// POUs/DIOC/F_GetVersion_FIXSUS_DIOC
FUNCTION F_GetVersion_FIXSUS_DIOC : INT(* Gets the library version info *)
VAR_INPUT
	nVersionElement		:	INT;
(*
	Possible nVersionElement parameter:
	1	:	major number
	2	:	minor number
	3	:	revision number
*)
END_VAR
(* Version history:
Date		|	Version				|	created with					|	Author				|	Remark
dd.mm.yyyy	|						|									|						|
-----------------------------------------------------------------------------------------------------------------------------------------------------------------------------------------------------------------------------------------------------------------------------------
23.12.2016	|	1.0.0				|	TCAT2.11 B2249					|	RK					|	first release
01.03.2017	|	2.0.0				|	TCAT2.11 B2249					|	FixSus				|	Array implementation, FB_Dioc
17.04.2017	|	2.1.0				|	TCAT2.11 B2249					|	RK					|	Library base
01.12.2017	|	3.5.0				|	TCAT2.11 B2259					|	FixSus				|	More generic implementation without arrays
26.01.2018	|	3.6.0				|	TCAT2.11 B2259					|	RK					|	General cleanup for final library and sample
26.01.2018	|	3.7.0				|	TCAT2.11 B2258					|	FixSus (AH)			|	Changed startup timer and visualisation RA
22.03.2018	|	3.8.0				|	TCAT2.11 B2258					|	FixSus (AH)			|	Added comments on visualisation RC
26.03.2018	|	3.9.0				|	TCAT2.11 B2258					|	FixSus (AH/HS)		|	Fixed bugs with DO 45,46 and 47 and added a 1 minute check on the input to know if the island is unplugged.
28.03.2018	|	3.10.0				|	TCAT2.11 B2258					|	FixSus (AH)			|	Added dewpoint calculation to the TP10 and deleted infrared measurements
17.04.2018	|	3.11.0				|	TCAT2.11 B2258					|	FixSus (AH)			| 	Added ForceSend Bools to the RC. If set to true, the analog values will be send immediatly.
19.06.2018	|	3.12.0				| 	TCAT2.11 B2258					|	FixSus (AH)			|	Added input to the TP10 to reset CO2/VOC sensor
19.06.2018	|	3.13.0				| 	TCAT2.11 B2258					|	FixSus (AH)			|	Fixed bug with buffer priority, small change to visualisations and added delay time to the RC startup list.
22.06.2018	|	3.14.0				| 	TCAT2.11 B2258					|	FixSus (AH)			|	VOC/eCO2 values are original sensor values again.
01.07.2018	|	3.15.0				|	TCAT2.11 B2258					|	FixSus (AH)			|	Updated startup timer
02.10.2018	|	3.16.0				|	TCAT2.11 B2258					|	FixSus (AH)			|	Added standard values to RC comments
13.03.2019	|	3.19.0				|	TCAT2.11 B2258					|	FixSus (AH)			|	Added version check to the VOC/eCO2 correction
28.05.2019	|	3.20.0				|	TCAT2.11 B2258					|	FixSus (AH)			|	Fixed startup list bug and sync message is the highest priority message now
30.08.2019	|	3.21.0				|	TCAT2.11 B2258					|	FixSus (AH) 		| 	Deleted reference to the currentvisu variable
12.03.2020	|	3.22.0				|	TCAT2.11 B2259					|	FixSus (AH)			|	RC intervals now use UDINT instead of INTS to avoid overflows with big timing intervals.
20.08.2020	|	3.23.0				|	TCAT2.11 B2277					| 	FixSus (AH)			| 	Completed RC descriptions in english.
27.10.2020	|	3.24.0				|	TCAT2.11 B2277					| 	FixSus (AH)			| 	TP10's with versions between 01/06/2020 and 08/10/2020 will send their temperature offset on a cyclic basis. Also deleted implicit conversions.
26.11.2020	|	3.25.0				|	TCAT2.11 B2277					|	FixSus (AH)			|	Sensitivity is now adjustable through the PLC program
*)

CASE nVersionElement OF
1:	(* major number *)
	F_GetVersion_FIXSUS_DIOC := 3;
2:	(* minor number *)
	F_GetVersion_FIXSUS_DIOC := 25;
3:	(* revision number *)
	F_GetVersion_FIXSUS_DIOC := 0;
ELSE
	F_GetVersion_FIXSUS_DIOC := -1;
END_CASE

END_FUNCTION

// Visualizations/DIOC/RC/RC_PARTS/RC_FP
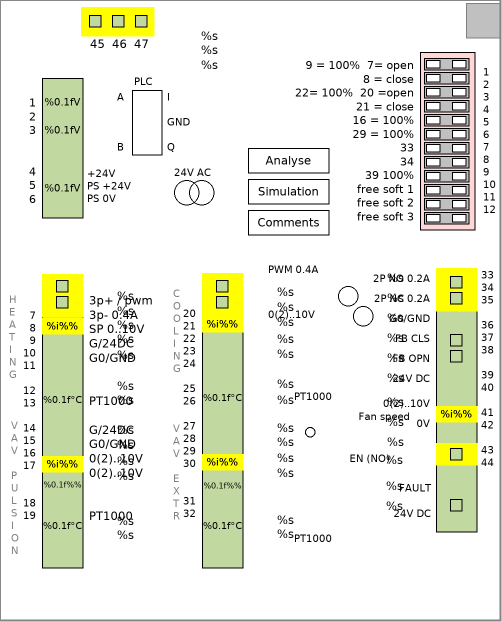
VISUALIZATION RC_FP  // 502x622
VAR_IN_OUT
	m_Input_GROUP : None;
END_VAR
    Rectangle (0,0 500x620)
    Rectangle (81,7 72x28)
    Rectangle (81,7 73x29), invisible if: NOT m_Input_GROUP._bSim, input disabled if: NOT m_Input_GROUP._bSim
    Rectangle (202,274 41x294)
    Rectangle (436,268 41x264)
    Rectangle (202,273 41x43), invisible if: NOT m_Input_GROUP._bSim, input disabled if: NOT m_Input_GROUP._bSim
    Rectangle (436,268 41x43), invisible if: NOT m_Input_GROUP._bSim, input disabled if: NOT m_Input_GROUP._bSim
    Rectangle (436,443 41x22), invisible if: NOT m_Input_GROUP._bSim, input disabled if: NOT m_Input_GROUP._bSim
    Rectangle (42,274 41x294)
    Rectangle (42,274 41x43), invisible if: NOT m_Input_GROUP._bSim, input disabled if: NOT m_Input_GROUP._bSim
    Polyline (133,133)
    Polyline (72,112)
    Rectangle (262,46 155x190), "9 = 100% 7= open 8 = close 22= 100% 20 =open 21 = close 16 = 100% 29 = 100% 33 34 39 100% free soft 1 free soft 2 free soft 3"
    Rectangle (24,268 15x295), "7 8 9 10 11 12 13 14 15 16 17 18 19"
    Rectangle (86,268 90x295), "3p+ / pwm 3p- 0.4A SP 0..10V G/24DC G0/GND PT1000 G/24DC G0/GND 0(2)..10V 0(2)..10V PT1000", invisible if: (m_Input_GROUP._bComments) <> 0
    Rectangle (184,266 15x295), "20 21 22 23 24 25 26 27 28 29 30 31 32"
    Rectangle (6,272 10x130), "H E A T I N G"
    Rectangle (8,416 10x144), "V A V P U L S I O N"
    Rectangle (170,411 10x135), "V A V E X T R"
    Rectangle (170,266 10x130), "C O O L I N G"
    Rectangle (42,392 41x16), "%0.1f°C", text variable: m_Input_GROUP.qfTempHeatingWater
    Rectangle (42,518 41x16), "%0.1f°C", text variable: m_Input_GROUP.qfTempAirPulsion
    Rectangle (42,318 41x16), "%i%%", text variable: m_Input_GROUP._iSpHeatingSim, invisible if: NOT m_Input_GROUP._bSim, input disabled if: NOT m_Input_GROUP._bSim
        OnMouseDown: write the text variable via VisuDialogs.Numpad, min 0, max 100
    Rectangle (42,456 41x16), "%i%%", text variable: m_Input_GROUP._iSpPulsionSim, invisible if: NOT m_Input_GROUP._bSim, input disabled if: NOT m_Input_GROUP._bSim
        OnMouseDown: write the text variable via VisuDialogs.Numpad, min 0, max 100
    Rectangle (42,477 41x16), "%0.1f%%", text variable: m_Input_GROUP.qfPulsionFB
    Rectangle (56,280 12x12), colour toggle: (m_Input_GROUP.bHeating_3P_plus) <> 0, invisible if: (m_Input_GROUP._bSim) <> 0, input disabled if: (m_Input_GROUP._bSim) <> 0
    Rectangle (56,296 12x12), colour toggle: (m_Input_GROUP.bHeating_3P_min) <> 0, invisible if: (m_Input_GROUP._bSim) <> 0, input disabled if: (m_Input_GROUP._bSim) <> 0
    Rectangle (202,390 41x16), "%0.1f°C", text variable: m_Input_GROUP.qfTempIceWater
    Rectangle (202,518 41x16), "%0.1f°C", text variable: m_Input_GROUP.qfTempAirExtraction
    Rectangle (202,316 41x16), "%i%%", text variable: m_Input_GROUP._iSpCoolingSim, invisible if: NOT m_Input_GROUP._bSim, input disabled if: NOT m_Input_GROUP._bSim
        OnMouseDown: write the text variable via VisuDialogs.Numpad, min 0, max 100
    Rectangle (202,454 41x16), "%i%%", text variable: m_Input_GROUP._iSpExtractionSim, invisible if: NOT m_Input_GROUP._bSim, input disabled if: NOT m_Input_GROUP._bSim
        OnMouseDown: write the text variable via VisuDialogs.Numpad, min 0, max 100
    Rectangle (202,478 41x16), "%0.1f%%", text variable: m_Input_GROUP.qfExtractionFB
    Rectangle (216,296 12x12), colour toggle: (m_Input_GROUP._bCooling_3P_minSim) <> 0, invisible if: NOT m_Input_GROUP._bSim, input disabled if: NOT m_Input_GROUP._bSim
        toggle m_Input_GROUP._bCooling_3P_minSim
    Rectangle (216,280 12x12), colour toggle: (m_Input_GROUP._bCooling_3P_plusSim) <> 0, invisible if: NOT m_Input_GROUP._bSim, input disabled if: NOT m_Input_GROUP._bSim
        toggle m_Input_GROUP._bCooling_3P_plusSim
    Rectangle (478,268 15x295), "33 34 35 36 37 38 39 40 41 42 43 44"
    Rectangle (436,406 41x16), "%i%%", text variable: m_Input_GROUP._iSpFanSim, invisible if: NOT m_Input_GROUP._bSim, input disabled if: NOT m_Input_GROUP._bSim
        OnMouseDown: write the text variable via VisuDialogs.Numpad, min 0, max 100
    Rectangle (450,276 12x12), colour toggle: (m_Input_GROUP._bFireDamper_OPNSim) <> 0, invisible if: NOT m_Input_GROUP._bSim, input disabled if: NOT m_Input_GROUP._bSim
        toggle m_Input_GROUP._bFireDamper_OPNSim
    Rectangle (450,292 12x12), colour toggle: (m_Input_GROUP._bFireDamper_CLSSim) <> 0, invisible if: NOT m_Input_GROUP._bSim, input disabled if: NOT m_Input_GROUP._bSim
        toggle m_Input_GROUP._bFireDamper_CLSSim
    Rectangle (450,350 12x12), colour toggle: (m_Input_GROUP.qbFireDamperFB_OPN) <> 0
    Rectangle (450,334 12x12), colour toggle: (m_Input_GROUP.qbFireDamperFB_CLS) <> 0
    Rectangle (450,448 12x12), colour toggle: (m_Input_GROUP._bEnableFanSim) <> 0, invisible if: NOT m_Input_GROUP._bSim, input disabled if: NOT m_Input_GROUP._bSim
        toggle m_Input_GROUP._bEnableFanSim
    Rectangle (24,83 15x150), "1 2 3 4 5 6"
    Rectangle (42,78 41x140)
    Rectangle (42,180 41x16), "%0.1fV", text variable: m_Input_GROUP.qfACVoltageLevel
    Rectangle (42,94 41x16), "%0.1fV", text variable: m_Input_GROUP.qrVoltageLevelA
    Rectangle (42,122 41x16), "%0.1fV", text variable: m_Input_GROUP.qrVoltageLevelB
    Rectangle (420,52 55x178)
    Rectangle (480,46 15x190), "1 2 3 4 5 6 7 8 9 10 11 12"
    Frame (424,58 47x14)
        shows UDO_DIPSWITCH(m_Input_GROUP := m_Input_GROUP, m_Input_ON_SIGNAAL := qarr_bDipSwitches[1])
    Frame (424,72 47x14)
        shows UDO_DIPSWITCH(m_Input_GROUP := m_Input_GROUP, m_Input_ON_SIGNAAL := qarr_bDipSwitches[2])
    Frame (424,86 47x14)
        shows UDO_DIPSWITCH(m_Input_GROUP := m_Input_GROUP, m_Input_ON_SIGNAAL := qarr_bDipSwitches[3])
    Frame (424,100 47x14)
        shows UDO_DIPSWITCH(m_Input_GROUP := m_Input_GROUP, m_Input_ON_SIGNAAL := qarr_bDipSwitches[4])
    Frame (424,114 47x14)
        shows UDO_DIPSWITCH(m_Input_GROUP := m_Input_GROUP, m_Input_ON_SIGNAAL := qarr_bDipSwitches[5])
    Frame (424,128 47x14)
        shows UDO_DIPSWITCH(m_Input_GROUP := m_Input_GROUP, m_Input_ON_SIGNAAL := qarr_bDipSwitches[6])
    Frame (424,142 47x14)
        shows UDO_DIPSWITCH(m_Input_GROUP := m_Input_GROUP, m_Input_ON_SIGNAAL := qarr_bDipSwitches[7])
    Frame (424,156 47x14)
        shows UDO_DIPSWITCH(m_Input_GROUP := m_Input_GROUP, m_Input_ON_SIGNAAL := qarr_bDipSwitches[8])
    Frame (424,170 47x14)
        shows UDO_DIPSWITCH(m_Input_GROUP := m_Input_GROUP, m_Input_ON_SIGNAAL := qarr_bDipSwitches[9])
    Frame (424,184 47x14)
        shows UDO_DIPSWITCH(m_Input_GROUP := m_Input_GROUP, m_Input_ON_SIGNAAL := qarr_bDipSwitches[10])
    Frame (424,198 47x14)
        shows UDO_DIPSWITCH(m_Input_GROUP := m_Input_GROUP, m_Input_ON_SIGNAAL := qarr_bDipSwitches[11])
    Frame (424,212 47x14)
        shows UDO_DIPSWITCH(m_Input_GROUP := m_Input_GROUP, m_Input_ON_SIGNAAL := qarr_bDipSwitches[12])
    Polyline (224,185)
    Polyline (224,200)
    Rectangle (132,90 30x65)
    Polyline (177,200)
    Polyline (164,210)
    Polyline (168,210)
    Ellipse (174,180 25x25)
    Ellipse (189,180 25x25)
    Rectangle (96,82 31x80), "A B"
    Rectangle (164,82 30x80), "I GND Q"
    Rectangle (131,74 40x15), "PLC"
    Rectangle (84,146 65x80), "+24V PS +24V PS 0V"
    Rectangle (144,165 70x15), "24V AC"
    Polyline (133,187)
    Polyline (111,171)
    Rectangle (248,179 81x25), "Simulation"
        toggle m_Input_GROUP._bSim
    Rectangle (56,280 12x12), colour toggle: (m_Input_GROUP._bHeating_3P_plusSim) <> 0, invisible if: NOT m_Input_GROUP._bSim, input disabled if: NOT m_Input_GROUP._bSim
        toggle m_Input_GROUP._bHeating_3P_plusSim
    Rectangle (56,296 12x12), colour toggle: (m_Input_GROUP._bHeating_3P_minSim) <> 0, invisible if: NOT m_Input_GROUP._bSim, input disabled if: NOT m_Input_GROUP._bSim
        toggle m_Input_GROUP._bHeating_3P_minSim
    Rectangle (42,318 41x16), "%i%%", text variable: m_Input_GROUP.iSpHeating, invisible if: (m_Input_GROUP._bSim) <> 0, input disabled if: (m_Input_GROUP._bSim) <> 0
    Rectangle (42,456 41x16), "%i%%", text variable: m_Input_GROUP.iSpPulsion, invisible if: (m_Input_GROUP._bSim) <> 0, input disabled if: (m_Input_GROUP._bSim) <> 0
    Rectangle (202,316 41x16), "%i%%", text variable: m_Input_GROUP.iSpCooling, invisible if: (m_Input_GROUP._bSim) <> 0, input disabled if: (m_Input_GROUP._bSim) <> 0
    Rectangle (202,454 41x16), "%i%%", text variable: m_Input_GROUP.iSpExtraction, invisible if: (m_Input_GROUP._bSim) <> 0, input disabled if: (m_Input_GROUP._bSim) <> 0
    Rectangle (216,296 12x12), colour toggle: (m_Input_GROUP.bCooling_3P_min) <> 0, invisible if: (m_Input_GROUP._bSim) <> 0, input disabled if: (m_Input_GROUP._bSim) <> 0
    Rectangle (216,280 12x12), colour toggle: (m_Input_GROUP.bCooling_3P_plus) <> 0, invisible if: (m_Input_GROUP._bSim) <> 0, input disabled if: (m_Input_GROUP._bSim) <> 0
    Rectangle (436,406 41x16), "%i%%", text variable: m_Input_GROUP.iSpFan, invisible if: (m_Input_GROUP._bSim) <> 0, input disabled if: (m_Input_GROUP._bSim) <> 0
    Rectangle (450,276 12x12), colour toggle: (m_Input_GROUP.bFireDamper_OPN) <> 0, invisible if: (m_Input_GROUP._bSim) <> 0, input disabled if: (m_Input_GROUP._bSim) <> 0
    Rectangle (450,292 12x12), colour toggle: (m_Input_GROUP.bFireDamper_CLS) <> 0, invisible if: (m_Input_GROUP._bSim) <> 0, input disabled if: (m_Input_GROUP._bSim) <> 0
    Rectangle (450,448 12x12), colour toggle: (m_Input_GROUP.bEnableFan) <> 0, invisible if: (m_Input_GROUP._bSim) <> 0, input disabled if: (m_Input_GROUP._bSim) <> 0
    Rectangle (450,499 12x12), colour toggle: (m_Input_GROUP.qbFanFault) <> 0
    Group (466,3 32x33)
        toggle m_Input_GROUP._bSelected
        RoundedRectangle (0,0 34x35)
        Polyline (28,28)
        Polyline (7,28)
    Rectangle (87,38 74x12), "45 46 47", invisible if: (m_Input_GROUP._bComments) <> 0
    Rectangle (89,15 12x12), colour toggle: (m_Input_GROUP.bRelais_45) <> 0, invisible if: (m_Input_GROUP._bSim) <> 0, input disabled if: (m_Input_GROUP._bSim) <> 0
    Rectangle (112,15 12x12), colour toggle: (m_Input_GROUP.bRelais_46) <> 0, invisible if: (m_Input_GROUP._bSim) <> 0, input disabled if: (m_Input_GROUP._bSim) <> 0
    Rectangle (135,15 12x12), colour toggle: (m_Input_GROUP.bRelais_47) <> 0, invisible if: (m_Input_GROUP._bSim) <> 0, input disabled if: (m_Input_GROUP._bSim) <> 0
    Rectangle (89,15 12x12), colour toggle: (m_Input_GROUP._bRelais_45Sim) <> 0, invisible if: NOT m_Input_GROUP._bSim, input disabled if: NOT m_Input_GROUP._bSim
        toggle m_Input_GROUP._bRelais_45Sim
    Rectangle (112,15 12x12), colour toggle: (m_Input_GROUP._bRelais_46Sim) <> 0, invisible if: NOT m_Input_GROUP._bSim, input disabled if: NOT m_Input_GROUP._bSim
        toggle m_Input_GROUP._bRelais_46Sim
    Rectangle (135,15 12x12), colour toggle: (m_Input_GROUP._bRelais_47Sim) <> 0, invisible if: NOT m_Input_GROUP._bSim, input disabled if: NOT m_Input_GROUP._bSim
        toggle m_Input_GROUP._bRelais_47Sim
    Rectangle (248,148 81x25), "Analyse", invisible if: NOT Global_DIOC_Variables_Debug.DIOC_Debug, input disabled if: NOT Global_DIOC_Variables_Debug.DIOC_Debug
        toggle m_Input_GROUP._bAnalyse
    Rectangle (248,210 81x25), "Comments"
        toggle m_Input_GROUP._bComments
    Group (245,262 192x291), invisible if: (m_Input_GROUP._bComments) <> 0
        Polyline (0,30)
        Polyline (0,105)
        Polyline (70,40)
        Polyline (70,30)
        Polyline (70,25)
        Polyline (70,35)
        Polyline (40,65)
        Polyline (40,70)
        Polyline (30,105)
        Group (26,6 18x33)
            Polygon (20,20)
            Polyline (20,20)
        Group (41,51 18x33)
            Polygon (20,20)
            Polyline (20,20)
        Polyline (40,120)
        Polyline (40,145)
        Polyline (40,263)
        Polyline (40,288)
        Polyline (50,214)
        Polyline (50,195)
        Polyline (50,205)
        Polyline (50,215)
        Polyline (80,180)
        Ellipse (60,165 10x10)
        Ellipse (93,24 20x20)
        Rectangle (20,0 60x15), "PWM 0.4A"
        Rectangle (20,45 60x15), "0(2)..10V"
        Rectangle (46,127 60x15), "PT1000"
        Rectangle (46,269 60x15), "PT1000"
        Ellipse (108,44 20x20)
        Polyline (193,24)
        Polyline (193,44)
        Polyline (193,64)
        Polyline (118,69)
        Polyline (193,124)
        Polyline (118,79)
        Polyline (118,99)
        Polyline (133,149)
        Polyline (133,169)
        Polyline (163,189)
        Polyline (118,204)
        Polyline (168,194)
        Polyline (178,189)
        Polyline (124,224)
        Polyline (194,259)
        Rectangle (118,9 70x15), "2P NO 0.2A"
        Rectangle (118,29 70x15), "2P NC 0.2A"
        Rectangle (118,49 70x15), "G0/GND"
        Rectangle (118,69 70x15), "FB CLS"
        Rectangle (118,89 70x15), "FB OPN"
        Rectangle (118,109 70x15), "24V DC"
        Rectangle (118,134 70x15), "0(2)..10V"
        Rectangle (98,147 70x15), "Fan speed"
        Rectangle (118,154 70x15), "0V"
        Rectangle (78,189 70x15), "EN (NO)"
        Rectangle (119,219 70x14), "FAULT"
        Rectangle (119,244 70x15), "24V DC"
        Polyline (50,215)
        Polyline (103,104)
        Polyline (17,220)
        Polyline (5,201)
    Rectangle (84,289 83x14), "%s", text variable: m_Input_GROUP.arr_sConnectionComments[1], invisible if: NOT m_Input_GROUP._bComments, input disabled if: NOT m_Input_GROUP._bComments
        OnMouseDown: write the text variable via Edit
    Rectangle (84,304 83x14), "%s", text variable: m_Input_GROUP.arr_sConnectionComments[2], invisible if: NOT m_Input_GROUP._bComments, input disabled if: NOT m_Input_GROUP._bComments
        OnMouseDown: write the text variable via Edit
    Rectangle (84,318 83x14), "%s", text variable: m_Input_GROUP.arr_sConnectionComments[3], invisible if: NOT m_Input_GROUP._bComments, input disabled if: NOT m_Input_GROUP._bComments
        OnMouseDown: write the text variable via Edit
    Rectangle (84,332 83x14), "%s", text variable: m_Input_GROUP.arr_sConnectionComments[4], invisible if: NOT m_Input_GROUP._bComments, input disabled if: NOT m_Input_GROUP._bComments
        OnMouseDown: write the text variable via Edit
    Rectangle (84,348 83x14), "%s", text variable: m_Input_GROUP.arr_sConnectionComments[5], invisible if: NOT m_Input_GROUP._bComments, input disabled if: NOT m_Input_GROUP._bComments
        OnMouseDown: write the text variable via Edit
    Rectangle (84,379 83x14), "%s", text variable: m_Input_GROUP.arr_sConnectionComments[6], invisible if: NOT m_Input_GROUP._bComments, input disabled if: NOT m_Input_GROUP._bComments
        OnMouseDown: write the text variable via Edit
    Rectangle (84,393 83x14), "%s", text variable: m_Input_GROUP.arr_sConnectionComments[7], invisible if: NOT m_Input_GROUP._bComments, input disabled if: NOT m_Input_GROUP._bComments
        OnMouseDown: write the text variable via Edit
    Rectangle (84,423 83x14), "%s", text variable: m_Input_GROUP.arr_sConnectionComments[8], invisible if: NOT m_Input_GROUP._bComments, input disabled if: NOT m_Input_GROUP._bComments
        OnMouseDown: write the text variable via Edit
    Rectangle (84,438 83x14), "%s", text variable: m_Input_GROUP.arr_sConnectionComments[9], invisible if: NOT m_Input_GROUP._bComments, input disabled if: NOT m_Input_GROUP._bComments
        OnMouseDown: write the text variable via Edit
    Rectangle (84,454 83x14), "%s", text variable: m_Input_GROUP.arr_sConnectionComments[10], invisible if: NOT m_Input_GROUP._bComments, input disabled if: NOT m_Input_GROUP._bComments
        OnMouseDown: write the text variable via Edit
    Rectangle (84,469 83x14), "%s", text variable: m_Input_GROUP.arr_sConnectionComments[11], invisible if: NOT m_Input_GROUP._bComments, input disabled if: NOT m_Input_GROUP._bComments
        OnMouseDown: write the text variable via Edit
    Rectangle (84,514 83x14), "%s", text variable: m_Input_GROUP.arr_sConnectionComments[12], invisible if: NOT m_Input_GROUP._bComments, input disabled if: NOT m_Input_GROUP._bComments
        OnMouseDown: write the text variable via Edit
    Rectangle (84,528 83x14), "%s", text variable: m_Input_GROUP.arr_sConnectionComments[13], invisible if: NOT m_Input_GROUP._bComments, input disabled if: NOT m_Input_GROUP._bComments
        OnMouseDown: write the text variable via Edit
    Rectangle (244,285 83x14), "%s", text variable: m_Input_GROUP.arr_sConnectionComments[14], invisible if: NOT m_Input_GROUP._bComments, input disabled if: NOT m_Input_GROUP._bComments
        OnMouseDown: write the text variable via Edit
    Rectangle (244,300 83x14), "%s", text variable: m_Input_GROUP.arr_sConnectionComments[15], invisible if: NOT m_Input_GROUP._bComments, input disabled if: NOT m_Input_GROUP._bComments
        OnMouseDown: write the text variable via Edit
    Rectangle (244,315 83x14), "%s", text variable: m_Input_GROUP.arr_sConnectionComments[16], invisible if: NOT m_Input_GROUP._bComments, input disabled if: NOT m_Input_GROUP._bComments
        OnMouseDown: write the text variable via Edit
    Rectangle (244,332 83x14), "%s", text variable: m_Input_GROUP.arr_sConnectionComments[17], invisible if: NOT m_Input_GROUP._bComments, input disabled if: NOT m_Input_GROUP._bComments
        OnMouseDown: write the text variable via Edit
    Rectangle (244,347 83x14), "%s", text variable: m_Input_GROUP.arr_sConnectionComments[18], invisible if: NOT m_Input_GROUP._bComments, input disabled if: NOT m_Input_GROUP._bComments
        OnMouseDown: write the text variable via Edit
    Rectangle (244,377 83x14), "%s", text variable: m_Input_GROUP.arr_sConnectionComments[19], invisible if: NOT m_Input_GROUP._bComments, input disabled if: NOT m_Input_GROUP._bComments
        OnMouseDown: write the text variable via Edit
    Rectangle (244,393 83x14), "%s", text variable: m_Input_GROUP.arr_sConnectionComments[20], invisible if: NOT m_Input_GROUP._bComments, input disabled if: NOT m_Input_GROUP._bComments
        OnMouseDown: write the text variable via Edit
    Rectangle (244,421 83x14), "%s", text variable: m_Input_GROUP.arr_sConnectionComments[21], invisible if: NOT m_Input_GROUP._bComments, input disabled if: NOT m_Input_GROUP._bComments
        OnMouseDown: write the text variable via Edit
    Rectangle (244,435 83x14), "%s", text variable: m_Input_GROUP.arr_sConnectionComments[22], invisible if: NOT m_Input_GROUP._bComments, input disabled if: NOT m_Input_GROUP._bComments
        OnMouseDown: write the text variable via Edit
    Rectangle (244,451 83x14), "%s", text variable: m_Input_GROUP.arr_sConnectionComments[23], invisible if: NOT m_Input_GROUP._bComments, input disabled if: NOT m_Input_GROUP._bComments
        OnMouseDown: write the text variable via Edit
    Rectangle (244,466 83x14), "%s", text variable: m_Input_GROUP.arr_sConnectionComments[24], invisible if: NOT m_Input_GROUP._bComments, input disabled if: NOT m_Input_GROUP._bComments
        OnMouseDown: write the text variable via Edit
    Rectangle (244,513 83x14), "%s", text variable: m_Input_GROUP.arr_sConnectionComments[25], invisible if: NOT m_Input_GROUP._bComments, input disabled if: NOT m_Input_GROUP._bComments
        OnMouseDown: write the text variable via Edit
    Rectangle (244,527 83x14), "%s", text variable: m_Input_GROUP.arr_sConnectionComments[26], invisible if: NOT m_Input_GROUP._bComments, input disabled if: NOT m_Input_GROUP._bComments
        OnMouseDown: write the text variable via Edit
    Rectangle (354,271 83x14), "%s", text variable: m_Input_GROUP.arr_sConnectionComments[27], invisible if: NOT m_Input_GROUP._bComments, input disabled if: NOT m_Input_GROUP._bComments
        OnMouseDown: write the text variable via Edit
    Rectangle (354,291 83x14), "%s", text variable: m_Input_GROUP.arr_sConnectionComments[28], invisible if: NOT m_Input_GROUP._bComments, input disabled if: NOT m_Input_GROUP._bComments
        OnMouseDown: write the text variable via Edit
    Rectangle (354,311 83x14), "%s", text variable: m_Input_GROUP.arr_sConnectionComments[29], invisible if: NOT m_Input_GROUP._bComments, input disabled if: NOT m_Input_GROUP._bComments
        OnMouseDown: write the text variable via Edit
    Rectangle (354,331 83x14), "%s", text variable: m_Input_GROUP.arr_sConnectionComments[30], invisible if: NOT m_Input_GROUP._bComments, input disabled if: NOT m_Input_GROUP._bComments
        OnMouseDown: write the text variable via Edit
    Rectangle (354,351 83x14), "%s", text variable: m_Input_GROUP.arr_sConnectionComments[31], invisible if: NOT m_Input_GROUP._bComments, input disabled if: NOT m_Input_GROUP._bComments
        OnMouseDown: write the text variable via Edit
    Rectangle (354,371 83x14), "%s", text variable: m_Input_GROUP.arr_sConnectionComments[32], invisible if: NOT m_Input_GROUP._bComments, input disabled if: NOT m_Input_GROUP._bComments
        OnMouseDown: write the text variable via Edit
    Rectangle (354,395 83x14), "%s", text variable: m_Input_GROUP.arr_sConnectionComments[33], invisible if: NOT m_Input_GROUP._bComments, input disabled if: NOT m_Input_GROUP._bComments
        OnMouseDown: write the text variable via Edit
    Rectangle (354,415 83x14), "%s", text variable: m_Input_GROUP.arr_sConnectionComments[34], invisible if: NOT m_Input_GROUP._bComments, input disabled if: NOT m_Input_GROUP._bComments
        OnMouseDown: write the text variable via Edit
    Rectangle (354,435 83x14), "%s", text variable: m_Input_GROUP.arr_sConnectionComments[35], invisible if: NOT m_Input_GROUP._bComments, input disabled if: NOT m_Input_GROUP._bComments
        OnMouseDown: write the text variable via Edit
    Rectangle (353,453 83x14), "%s", text variable: m_Input_GROUP.arr_sConnectionComments[36], invisible if: NOT m_Input_GROUP._bComments, input disabled if: NOT m_Input_GROUP._bComments
        OnMouseDown: write the text variable via Edit
    Rectangle (353,479 83x14), "%s", text variable: m_Input_GROUP.arr_sConnectionComments[37], invisible if: NOT m_Input_GROUP._bComments, input disabled if: NOT m_Input_GROUP._bComments
        OnMouseDown: write the text variable via Edit
    Rectangle (353,499 83x14), "%s", text variable: m_Input_GROUP.arr_sConnectionComments[38], invisible if: NOT m_Input_GROUP._bComments, input disabled if: NOT m_Input_GROUP._bComments
        OnMouseDown: write the text variable via Edit
    Rectangle (168,29 83x14), "%s", text variable: m_Input_GROUP.arr_sConnectionComments[39], invisible if: NOT m_Input_GROUP._bComments, input disabled if: NOT m_Input_GROUP._bComments
        OnMouseDown: write the text variable via Edit
    Rectangle (168,43 83x14), "%s", text variable: m_Input_GROUP.arr_sConnectionComments[40], invisible if: NOT m_Input_GROUP._bComments, input disabled if: NOT m_Input_GROUP._bComments
        OnMouseDown: write the text variable via Edit
    Rectangle (168,58 83x14), "%s", text variable: m_Input_GROUP.arr_sConnectionComments[41], invisible if: NOT m_Input_GROUP._bComments, input disabled if: NOT m_Input_GROUP._bComments
        OnMouseDown: write the text variable via Edit
    Polyline (190,45), invisible if: NOT m_Input_GROUP._bComments
    Polyline (190,56), invisible if: NOT m_Input_GROUP._bComments
    Polyline (190,68), invisible if: NOT m_Input_GROUP._bComments
END_VISUALIZATION

// Visualizations/DIOC/RC/RC_PARTS/RC_ROOM_ICON
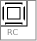
VISUALIZATION RC_ROOM_ICON  // 37x41
    Rectangle (0,0 27x26)
    Rectangle (7,7 13x12)
    Rectangle (5,3 17x0)
    Rectangle (5,23 17x0)
    Rectangle (24,6 0x14)
    Rectangle (3,6 0x14)
    Rectangle (-10,26 45x13), "RC"
    Rectangle (-2,0 30x25)
END_VISUALIZATION

// Visualizations/DIOC/RC/RC_PARTS/UDO_DIPSWITCH
VISUALIZATION UDO_DIPSWITCH  // 47x14
VAR_INPUT
	m_Input_GROUP : None;
END_VAR
VAR_INPUT
	m_Input_ON_SIGNAAL : None;
END_VAR
    Rectangle (0,0 45x12)
    Rectangle (28,2 14x8), invisible if: NOT m_Input_GROUP.m_Input_ON_SIGNAAL
    Rectangle (2,2 14x8), invisible if: ((m_Input_GROUP.m_Input_ON_SIGNAAL)) <> 0
END_VISUALIZATION

// Visualizations/DIOC/RC/RC
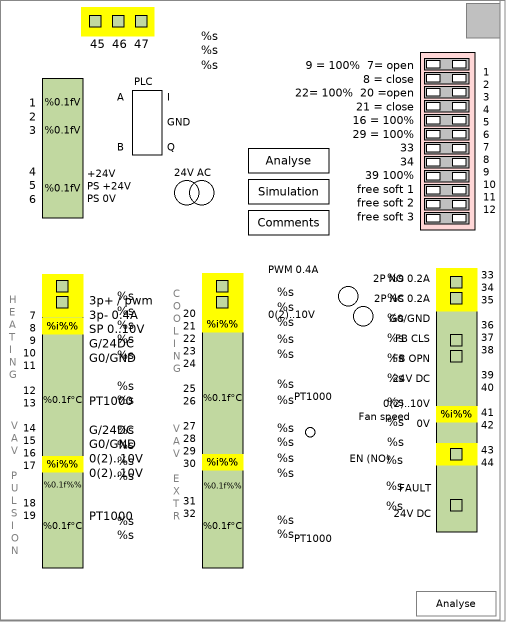
VISUALIZATION RC  // 506x622
VAR_IN_OUT
	m_Input_FB_RC : None;
END_VAR
VAR_IN_OUT
	m_Input_GROUP : None;
END_VAR
VAR_IN_OUT
	m_Input_AnalyseScherm : None;
END_VAR
    Frame (0,0 504x620)
        shows RC_FP(m_Input_GROUP := m_Input_FB_RC)
    Rectangle (416,591 80x25), "Analyse", invisible if: NOT Global_DIOC_Variables_Debug.DIOC_Debug, input disabled if: NOT Global_DIOC_Variables_Debug.DIOC_Debug
        toggle m_Input_GROUP._bAnalyse
END_VISUALIZATION

// Visualizations/DIOC/RC/RC_MINI
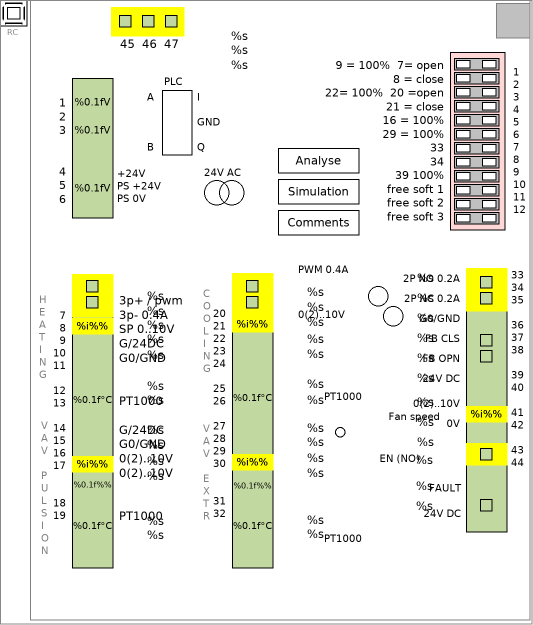
VISUALIZATION RC_MINI  // 533x625
VAR_IN_OUT
	m_Input_FB_RC : None;
END_VAR
VAR_IN_OUT
	m_Input_X_OFFSET : None;
END_VAR
VAR_IN_OUT
	m_Input_Y_OFFSET : None;
END_VAR
    Frame (0,0 27x33)
        shows RC_ROOM_ICON()
        toggle m_Input_FB_RC._bSelected
    Frame (30,0 501x623), invisible if: NOT (m_Input_FB_RC._bSelected), input disabled if: NOT (m_Input_FB_RC._bSelected)
        shows RC_FP(m_Input_GROUP := m_Input_FB_RC)
        p3560616238: m_Input_X_OFFSET
        p2738717112: m_Input_Y_OFFSET
END_VISUALIZATION

// Visualizations/DIOC/TP10/TP10_PARTS/TP10_FP
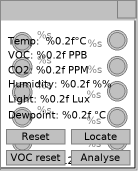
VISUALIZATION TP10_FP  // 138x171
VAR_IN_OUT
	m_Input_GROUP : None;
END_VAR
    Rectangle (0,18 135x150)
    Rectangle (0,-2 135x170)
    Rectangle (0,-2 135x22)
    Polygon (85,13), invisible if: (m_Input_GROUP.bRoomAnalyser) <> 0, input disabled if: (m_Input_GROUP.bRoomAnalyser) <> 0
    Polygon (99,13), invisible if: (m_Input_GROUP.bRoomAnalyser) <> 0, input disabled if: (m_Input_GROUP.bRoomAnalyser) <> 0
    Rectangle (92,-1 22x19), invisible if: (m_Input_GROUP.bRoomAnalyser) <> 0, input disabled if: (m_Input_GROUP.bRoomAnalyser) <> 0
        toggle m_Input_GROUP._bNextVisu
    Group (117,-1 17x17)
        toggle m_Input_GROUP._bSelected
        RoundedRectangle (0,0 19x19)
        Polyline (15,15)
        Polyline (3,15)
    Rectangle (68,0 22x19), invisible if: (m_Input_GROUP.bRoomAnalyser) <> 0, input disabled if: (m_Input_GROUP.bRoomAnalyser) <> 0
        toggle m_Input_GROUP._bPrevVisu
    Group (3,23 130x144), invisible if: m_Input_GROUP._iVis <> 0, input disabled if: m_Input_GROUP._iVis <> 0
        Rectangle (0,129 132x17), "%0.2f°C", text variable: m_Input_GROUP.qfRoomTemperature
        Group (8,101 78x26)
            Ellipse (1,8 20x20), colour variable: m_Input_GROUP._dwVisColor
            Ellipse (3,10 16x16), colour toggle: (m_Input_GROUP.arr_bLeds[5]) <> 0
            Rectangle (23,0 57x22), "%s", text variable: m_Input_GROUP.arr_sButtonComments[5]
            Rectangle (0,7 51x21), invisible if: (m_Input_GROUP.arr_bMasks[5]) <> 0, input disabled if: (m_Input_GROUP.arr_bMasks[5]) <> 0
                tap m_Input_GROUP._arr_bVisuButtons[5]
        Group (8,76 78x26)
            Ellipse (1,8 20x20), colour variable: m_Input_GROUP._dwVisColor
            Ellipse (3,10 16x16), colour toggle: (m_Input_GROUP.arr_bLeds[4]) <> 0
            Rectangle (23,0 57x22), "%s", text variable: m_Input_GROUP.arr_sButtonComments[4]
            Rectangle (0,7 51x21), invisible if: (m_Input_GROUP.arr_bMasks[4]) <> 0, input disabled if: (m_Input_GROUP.arr_bMasks[4]) <> 0
                tap m_Input_GROUP._arr_bVisuButtons[4]
        Group (9,51 77x26)
            Ellipse (0,8 20x20), colour variable: m_Input_GROUP._dwVisColor
            Ellipse (2,10 16x16), colour toggle: (m_Input_GROUP.arr_bLeds[3]) <> 0
            Rectangle (22,0 57x22), "%s", text variable: m_Input_GROUP.arr_sButtonComments[3]
            Rectangle (0,7 51x21), invisible if: (m_Input_GROUP.arr_bMasks[3]) <> 0, input disabled if: (m_Input_GROUP.arr_bMasks[3]) <> 0
                tap m_Input_GROUP._arr_bVisuButtons[3]
        Group (9,26 77x26)
            Ellipse (0,8 20x20), colour variable: m_Input_GROUP._dwVisColor
            Ellipse (2,10 16x16), colour toggle: (m_Input_GROUP.arr_bLeds[2]) <> 0
            Rectangle (22,0 57x22), "%s", text variable: m_Input_GROUP.arr_sButtonComments[2]
            Rectangle (0,7 51x21), invisible if: (m_Input_GROUP.arr_bMasks[2]) <> 0, input disabled if: (m_Input_GROUP.arr_bMasks[2]) <> 0
                tap m_Input_GROUP._arr_bVisuButtons[2]
        Group (46,7 78x23)
            Ellipse (58,0 20x20), colour variable: m_Input_GROUP._dwVisColor
            Ellipse (60,2 16x16), colour toggle: (m_Input_GROUP.arr_bLeds[6]) <> 0
            Rectangle (0,2 56x23), "%s", text variable: m_Input_GROUP.arr_sButtonComments[6]
            Rectangle (28,1 52x20), invisible if: (m_Input_GROUP.arr_bMasks[6]) <> 0, input disabled if: (m_Input_GROUP.arr_bMasks[6]) <> 0
                tap m_Input_GROUP._arr_bVisuButtons[6]
        Group (46,33 77x23)
            Ellipse (58,0 20x20), colour variable: m_Input_GROUP._dwVisColor
            Ellipse (60,2 16x16), colour toggle: (m_Input_GROUP.arr_bLeds[7]) <> 0
            Rectangle (0,2 56x23), "%s", text variable: m_Input_GROUP.arr_sButtonComments[7]
            Rectangle (27,1 52x20), invisible if: (m_Input_GROUP.arr_bMasks[7]) <> 0, input disabled if: (m_Input_GROUP.arr_bMasks[7]) <> 0
                tap m_Input_GROUP._arr_bVisuButtons[7]
        Group (45,58 79x23)
            Ellipse (59,0 20x20), colour variable: m_Input_GROUP._dwVisColor
            Ellipse (61,2 16x16), colour toggle: (m_Input_GROUP.arr_bLeds[8]) <> 0
            Rectangle (0,2 56x23), "%s", text variable: m_Input_GROUP.arr_sButtonComments[8]
            Rectangle (29,1 52x20), invisible if: (m_Input_GROUP.arr_bMasks[8]) <> 0, input disabled if: (m_Input_GROUP.arr_bMasks[8]) <> 0
                tap m_Input_GROUP._arr_bVisuButtons[8]
        Group (45,84 80x23)
            Ellipse (59,0 20x20), colour variable: m_Input_GROUP._dwVisColor
            Ellipse (61,2 16x16), colour toggle: (m_Input_GROUP.arr_bLeds[9]) <> 0
            Rectangle (0,2 56x23), "%s", text variable: m_Input_GROUP.arr_sButtonComments[9]
            Rectangle (30,0 52x20), invisible if: (m_Input_GROUP.arr_bMasks[9]) <> 0, input disabled if: (m_Input_GROUP.arr_bMasks[9]) <> 0
                tap m_Input_GROUP._arr_bVisuButtons[9]
        Group (45,108 79x22)
            Ellipse (59,0 20x20), colour variable: m_Input_GROUP._dwVisColor
            Ellipse (61,2 16x16), colour toggle: (m_Input_GROUP.arr_bLeds[10]) <> 0
            Rectangle (0,1 56x23), "%s", text variable: m_Input_GROUP.arr_sButtonComments[10]
            Rectangle (29,0 52x20), invisible if: (m_Input_GROUP.arr_bMasks[10]) <> 0, input disabled if: (m_Input_GROUP.arr_bMasks[10]) <> 0
                tap m_Input_GROUP._arr_bVisuButtons[10]
        Group (9,1 77x26)
            Ellipse (0,8 20x20), colour variable: m_Input_GROUP._dwVisColor
                p3450524324: m_Input_GROUP._dwVisColor
            Ellipse (2,10 16x16), colour toggle: (m_Input_GROUP.arr_bLeds[1]) <> 0
            Rectangle (22,0 57x22), "%s", text variable: m_Input_GROUP.arr_sButtonComments[1]
            Rectangle (0,7 51x21), invisible if: (m_Input_GROUP.arr_bMasks[1]) <> 0, input disabled if: (m_Input_GROUP.arr_bMasks[1]) <> 0
                tap m_Input_GROUP._arr_bVisuButtons[1]
    Group (5,33 126x130), invisible if: m_Input_GROUP._iVis <> 1, input disabled if: m_Input_GROUP._iVis <> 1
        Rectangle (0,0 128x16), "Temp: %0.2f°C", text variable: m_Input_GROUP.qfRoomTemperature
        Rectangle (0,14 128x16), "VOC: %0.2f PPB", text variable: m_Input_GROUP.qfVOC
        Rectangle (0,29 128x16), "CO2: %0.2f PPM", text variable: m_Input_GROUP.qfCO2
        Rectangle (0,43 128x16), "Humidity: %0.2f %%", text variable: m_Input_GROUP.qfHumidity
        Rectangle (0,58 128x16), "Light: %0.2f Lux", text variable: m_Input_GROUP.qfLux
        Rectangle (1,96 59x15), "Reset"
            toggle m_Input_GROUP.bReset
        Rectangle (66,117 59x15), "Analyse", invisible if: NOT Global_DIOC_Variables_Debug.DIOC_Debug, input disabled if: NOT Global_DIOC_Variables_Debug.DIOC_Debug
            toggle m_Input_GROUP._bAnalyse
        Rectangle (66,96 59x15), "Locate"
            toggle m_Input_GROUP.bLocate
        Rectangle (0,74 128x16), "Dewpoint: %0.2f °C", text variable: m_Input_GROUP.qfDewpoint
        Rectangle (1,117 59x15), "VOC reset"
            toggle m_Input_GROUP.bResetVOC
END_VISUALIZATION

// Visualizations/DIOC/TP10/TP10_PARTS/TP10_ROOM_ICON
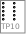
VISUALIZATION TP10_ROOM_ICON  // 26x34
    Ellipse (2,2 2x2)
    Ellipse (2,6 2x2)
    Ellipse (2,10 2x2)
    Ellipse (2,14 2x2)
    Ellipse (2,18 2x2)
    Ellipse (13,2 2x2)
    Ellipse (13,6 2x2)
    Ellipse (13,10 2x2)
    Ellipse (13,14 2x2)
    Ellipse (13,18 2x2)
    Rectangle (-5,0 29x32)
    Rectangle (-2,21 21x10), "TP10"
    Polyline (18,22)
END_VISUALIZATION

// Visualizations/DIOC/TP10/TP10
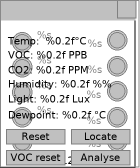
VISUALIZATION TP10  // 140x168
VAR_IN_OUT
	m_Input_ArrayNr : None;
END_VAR
VAR_IN_OUT
	m_Input_FB_TP10 : None;
END_VAR
    Frame (0,0 138x166)
        shows TP10_FP(m_Input_GROUP := m_Input_FB_TP10)
END_VISUALIZATION

// Visualizations/DIOC/TP10/TP10_MINI
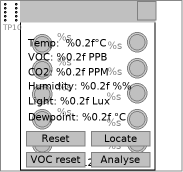
VISUALIZATION TP10_MINI  // 183x172
VAR_IN_OUT
	m_Input_X_OFFSET : None;
END_VAR
VAR_IN_OUT
	m_Input_Y_OFFSET : None;
END_VAR
VAR_IN_OUT
	m_Input_FB_TP10 : None;
END_VAR
    Frame (20,2 161x168), invisible if: NOT (m_Input_FB_TP10._bSelected), input disabled if: NOT (m_Input_FB_TP10._bSelected)
        shows TP10_FP(m_Input_GROUP := m_Input_FB_TP10)
        p3560616238: m_Input_X_OFFSET
        p2738717112: m_Input_Y_OFFSET
    Group (-5,1 27x30)
        toggle m_Input_FB_TP10._bSelected
        Ellipse (9,2 2x2)
        Ellipse (9,6 2x2)
        Ellipse (9,10 2x2)
        Ellipse (9,14 2x2)
        Ellipse (9,18 2x2)
        Ellipse (20,2 2x2)
        Ellipse (20,6 2x2)
        Ellipse (20,10 2x2)
        Ellipse (20,14 2x2)
        Ellipse (20,18 2x2)
        Rectangle (0,0 29x32)
        Rectangle (5,21 21x10), "TP10"
        Polyline (25,22)
END_VISUALIZATION
